FUNCTION_BLOCK FB_CommandChangeProduction EXTENDS FB_CommandChange IMPLEMENTS ITF_CommandChange
VAR

END_VAR

METHOD Execute : BOOL
VAR_INPUT
END_VAR
END_METHOD

METHOD FB_init : BOOL
VAR_INPUT
	bInitRetains : BOOL; // if TRUE, the retain variables are initialized (warm start / cold start)
	bInCopyCode : BOOL;  // if TRUE, the instance afterwards gets moved into the copy code (online change)
END_VAR
THIS^.SetText (eLocation := E_BaseLocation.pl, wsDescription := "Command change mode - Production");
THIS^.SetText (eLocation := E_BaseLocation.en, wsDescription := "Command change mode - Production");
THIS^.SetText (eLocation := E_BaseLocation.de, wsDescription := "Command change mode - Production");
THIS^.SetName (stName := THIS^.GetTexts ());
END_METHOD

END_FUNCTION_BLOCK

(* stored: Version 1.1.0.1
   POU FB_CommandChangeProduction: Id {955c8aa3-64ca-02f4-2f29-c4bdfe418e05}, SpecialFunc None
   Method Execute: Id {e331c9f4-9d24-0168-26da-d17c662e041c}
   Method FB_init: Id {65e40685-0b17-0852-253c-e218ec5fd955} *)
